// TIA Portal project "FactoryIO_Template_S7-1200_V16_V16" (V16)
// Vorlageprojekt für das Buch mit Zielsystem S7-1200

(* hardware
DEVICE "S7-1200-Station_1"  S7-1200 Station
   slot 0: "Baugruppenträger_0"  Rack  V1.0
   slot 1: "PLC_1"  CPU 1211C DC/DC/DC  6ES7 211-1AE40-0XB0  V4.1
*)

// ===== PLC "PLC_1"  CPU 1211C DC/DC/DC =====

VAR_GLOBAL   // PLC tag table "Standard-Variablentabelle"
   "belt 2m" AT %A0.0 : Bool;
   "start" AT %E0.0 : Bool;
   "stop" AT %E0.1 : Bool;
   "Tag_4" AT %I10.0 : Bool;
   "Tag_5" AT %Q10.0 : Bool;
   "Tag_6" AT %I10.1 : Bool;
   "belt 6m" AT %Q0.1 : Bool;
   "belt 4m" AT %Q0.2 : Bool;
   "elevator up" AT %Q0.3 : Bool;
   "inductive sensor 2" AT %I0.5 : Bool;
   "elevator left limit" AT %I0.3 : Bool;
   "elevator right limit" AT %I0.2 : Bool;
   "inductive sensor 1" AT %I0.4 : Bool;
   "elevator +" AT %Q0.5 : Bool;
   "down" AT %Q0.4 : Bool;
   "Tag_1" AT %M0.1 : Bool;
   "x" AT %M0.0 : Bool;
END_VAR

FUNCTION "MHJ-PLC-Lab-Function-S71200" : Void   // FC9000, SCL
{ S7_Optimized_Access := 'TRUE' }
VERSION : 0.1
   VAR_TEMP
      rdTimeReturn : Int;
      outputTime : DTL;
      SyncVal : Byte;
      forVal : Int;
      forVal_2 : Int;
      Value : Byte;
   END_VAR
   VAR CONSTANT
      CompVal : Byte := 16#34;
      Value_01 : Byte := 16#11;
      Value_01_DW : DWord := 16#A165_D992;
      Value_02_DW : DWord := 16#58BE_4401;
   END_VAR
BEGIN

   #Value:=PEEK(area := 16#82,
        dbNumber := 0,
        byteOffset := 511);
   #Value := #Value + 1;

   POKE(area := 16#82,
        dbNumber := 0,
        byteOffset := 511,
        value := #Value);

   POKE(area:=16#81,
        dbNumber:=0,
        byteOffset:=1016,
        value:=#Value_01_DW);
   POKE(area := 16#81,
        dbNumber := 0,
        byteOffset := 1020,
        value := #Value_02_DW);

   POKE(area := 16#81,
        dbNumber := 0,
        byteOffset := 511,
        value := B#16#00);

   FOR #forVal := 0 TO 120 DO
       FOR #forVal_2:=0 TO 10 DO
           #rdTimeReturn:=RD_SYS_T(#outputTime);
           #rdTimeReturn := WR_SYS_T(#outputTime);
           #rdTimeReturn := RD_SYS_T(#outputTime);
           #rdTimeReturn := WR_SYS_T(#outputTime);
       END_FOR;
       #SyncVal:= PEEK(area := 16#81,
                      dbNumber := 0,
                      byteOffset := 511);
       IF #SyncVal = #CompVal THEN
          GOTO M_1;
       END_IF;
   END_FOR;
   RETURN;

   M_1:
   POKE(area := 16#81,
        dbNumber := 0,
        byteOffset := 511,
        value := B#16#0);
END_FUNCTION

ORGANIZATION_BLOCK "Main"   // OB1, LAD, ProgramCycle
TITLE = "Main Program Sweep (Cycle)"
{ S7_Optimized_Access := 'TRUE' }
VERSION : 0.1
   VAR_INPUT
      Initial_Call : Bool;   // Initial call of this OB
      Remanence : Bool;   // =True, if remanent data are available
   END_VAR
BEGIN

REGION Network 1: Konnektierungsbaustein für PLC-Lab
   // Im Netzwerk 1 wird der Konnektierungsbaustein für PLC-Lab aufgerufen.
   // Dieser Aufruf darf nicht entfernt werden!
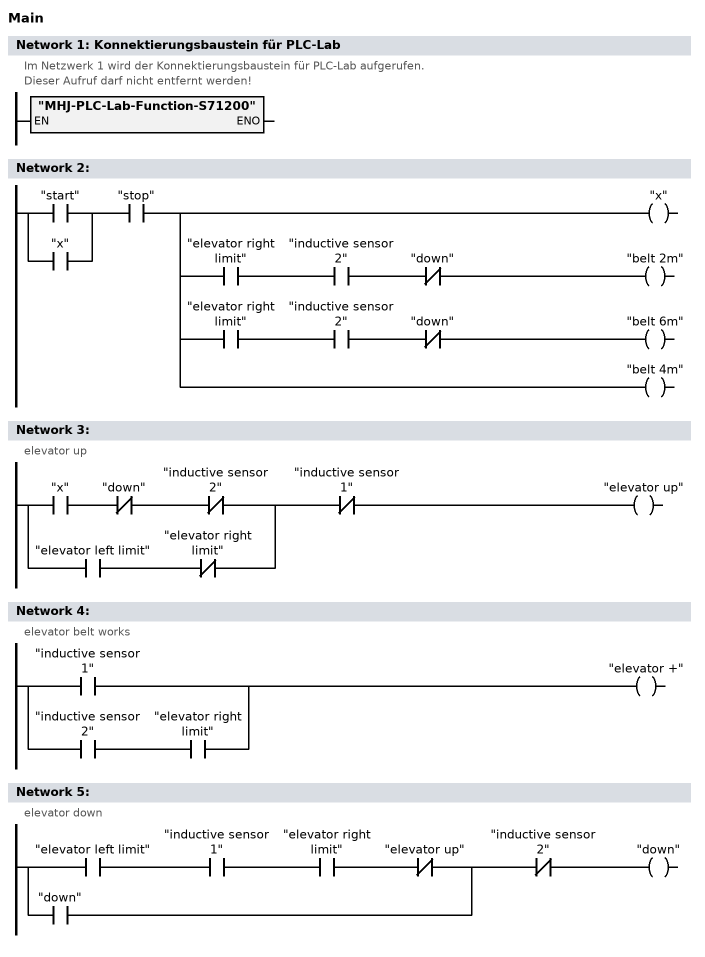
   RUNG wire#powerrail
      "MHJ-PLC-Lab-Function-S71200"()
   END_RUNG
   // the same network as SCL:
   "MHJ-PLC-Lab-Function-S71200"();
END_REGION

REGION Network 2
   RUNG wire#powerrail
      Contact( "start" )
      wire#w1
      Contact( "stop" )
      wire#w2
      Coil( "x" )
   END_RUNG
   RUNG wire#powerrail
      Contact( "x" )
   END_RUNG wire#w1
   RUNG wire#w2
      Contact( "elevator right limit" )
      Contact( "inductive sensor 2" )
      I_Contact( "down" )
      Coil( "belt 2m" )
   END_RUNG
   RUNG wire#w2
      Contact( "elevator right limit" )
      Contact( "inductive sensor 2" )
      I_Contact( "down" )
      Coil( "belt 6m" )
   END_RUNG
   RUNG wire#w2
      Coil( "belt 4m" )
   END_RUNG
   // the same network as SCL:
   "x" := ("start" OR "x") AND "stop";
   "belt 2m" := "x" AND "elevator right limit" AND "inductive sensor 2" AND NOT "down";
   "belt 6m" := "x" AND "elevator right limit" AND "inductive sensor 2" AND NOT "down";
   "belt 4m" := "x";
END_REGION

REGION Network 3
   // elevator up
   RUNG wire#powerrail
      Contact( "x" )
      I_Contact( "down" )
      I_Contact( "inductive sensor 2" )
      wire#w1
      I_Contact( "inductive sensor 1" )
      Coil( "elevator up" )
   END_RUNG
   RUNG wire#powerrail
      Contact( "elevator left limit" )
      I_Contact( "elevator right limit" )
   END_RUNG wire#w1
   // the same network as SCL:
   "elevator up" := (("x" AND NOT "down" AND NOT "inductive sensor 2") OR ("elevator left limit" AND NOT "elevator right limit")) AND NOT "inductive sensor 1";
END_REGION

REGION Network 4
   // elevator belt works
   RUNG wire#powerrail
      Contact( "inductive sensor 1" )
      wire#w1
      Coil( "elevator +" )
   END_RUNG
   RUNG wire#powerrail
      Contact( "inductive sensor 2" )
      Contact( "elevator right limit" )
   END_RUNG wire#w1
   // the same network as SCL:
   "elevator +" := "inductive sensor 1" OR ("inductive sensor 2" AND "elevator right limit");
END_REGION

REGION Network 5
   // elevator down
   RUNG wire#powerrail
      Contact( "elevator left limit" )
      Contact( "inductive sensor 1" )
      Contact( "elevator right limit" )
      I_Contact( "elevator up" )
      wire#w1
      I_Contact( "inductive sensor 2" )
      Coil( "down" )
   END_RUNG
   RUNG wire#powerrail
      Contact( "down" )
   END_RUNG wire#w1
   // the same network as SCL:
   "down" := (("elevator left limit" AND "inductive sensor 1" AND "elevator right limit" AND NOT "elevator up") OR "down") AND NOT "inductive sensor 2";
END_REGION
END_ORGANIZATION_BLOCK